Omron CX-Programmer project 新工程 (CX-Programmer 9.73)

# PLC 新PLC1: CPM1(CPM1A) CPU30

## Global symbols (name address type ; comment)
10.00 BOOL  ; KUP
10.01 BOOL  ; KDN
CNT012 BOOL  ; 50

## Program 新程序1 (no task)
; 项目信息： / 这是一个商场中的自动扶梯控制系统，使用欧姆龙 PLC 控制器 CPM1(CPM1A) CPU30 实现。 / 系统通过启动按钮启动扶梯运行，只有在停止按钮未按下时才能启动。 / 操作人员通过上行按钮和下行按钮选择运行方向，上行模式和下行模式不能同时为真。 / 在扶梯运行过程中，操作人员不能手动控制扶梯方向。 / 设备信息： / 系统使用PLC控制器CPM1(CPM1A) CPU30进行控制。 / 硬件包括启动按钮、上行按钮、下行按钮、停止按钮、安全传感器、速度传感器、故障信号输入和报警灯。 / 预期控制： / 系统通过启动按钮和运行使能启动扶梯运行，运行使能由停止按钮2控制。 / 操作人员通过上行按钮和下行按钮选择运行方向，分别激活上行控制或下行控制。 / 上行控制和下行控制通过互锁逻辑设计，尝试避免同时激活。 / 扶梯运行时，安全传感器1-5和速度传感器实时监控状态。 / 安全传感器5检测到异常时，通过计数器记录，若计数器值小于50，设置标志。 / 速度传感器检测到速度异常时，置位速度异常标志。 / 故障信号1-6触发时，置位故障标志1-6。 / 故障信号1触发时，置位故障标志1，记录故障状态。 / 在扶梯运行过程中，方向选择受定时器和标志控制。 / 停止按钮1和停止按钮2可影响扶梯运行，具体逻辑由定时器和内部标志控制。 / 手动/自动切换开关允许操作人员灵活选择控制模式，运行状态输出则向外部设备反馈扶梯运行状态。

### Section 段1

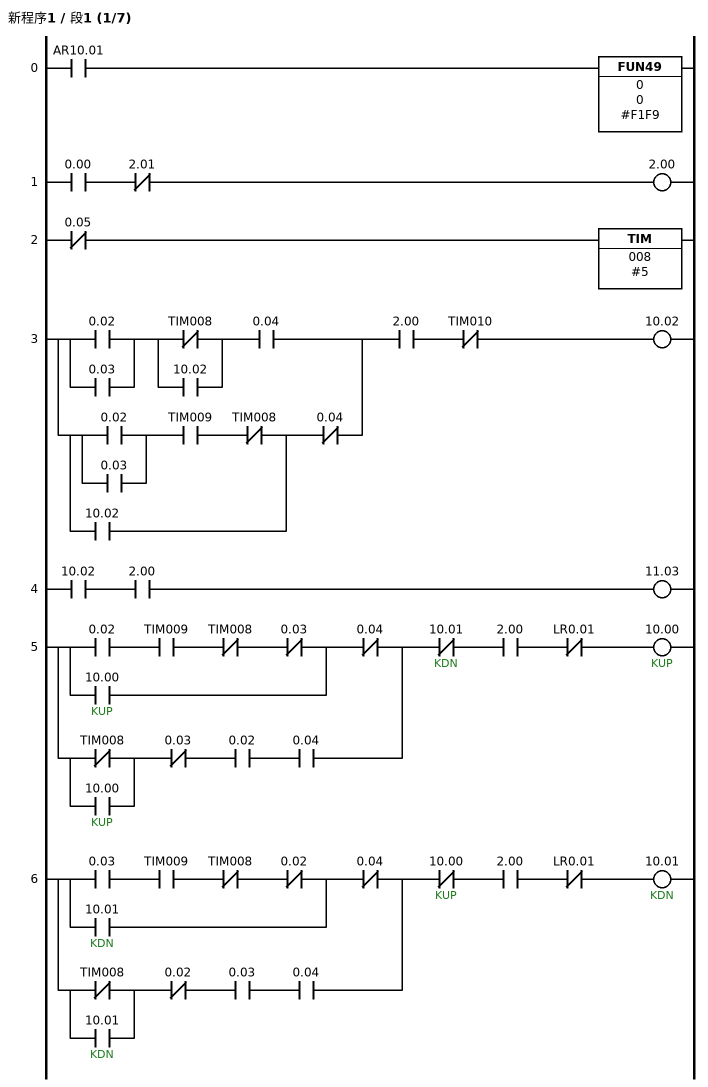
; rung 0
LD AR10.01
FUN49 0 0 #F1F9
; rung 1
LD 0.00
ANDNOT 2.01
OUT 2.00
; rung 2
LDNOT 0.05
TIM 008 #5
; rung 3
LD 0.02
OR 0.03
LDNOT TIM008
OR 10.02
ANDLD
AND 0.04
LD 0.02
OR 0.03
AND TIM009
ANDNOT TIM008
OR 10.02
ANDNOT 0.04
ORLD
AND 2.00
ANDNOT TIM010
OUT 10.02
; rung 4
LD 10.02
AND 2.00
OUT 11.03
; rung 5
LD 0.02
AND TIM009
ANDNOT TIM008
ANDNOT 0.03
OR 10.00  ; KUP
ANDNOT 0.04
LDNOT TIM008
OR 10.00  ; KUP
ANDNOT 0.03
AND 0.02
AND 0.04
ORLD
ANDNOT 10.01  ; KDN
AND 2.00
ANDNOT LR0.01
OUT 10.00  ; KUP
; rung 6
LD 0.03
AND TIM009
ANDNOT TIM008
ANDNOT 0.02
OR 10.01  ; KDN
ANDNOT 0.04
LDNOT TIM008
OR 10.01  ; KDN
ANDNOT 0.02
AND 0.03
AND 0.04
ORLD
ANDNOT 10.00  ; KUP
AND 2.00
ANDNOT LR0.01
OUT 10.01  ; KDN

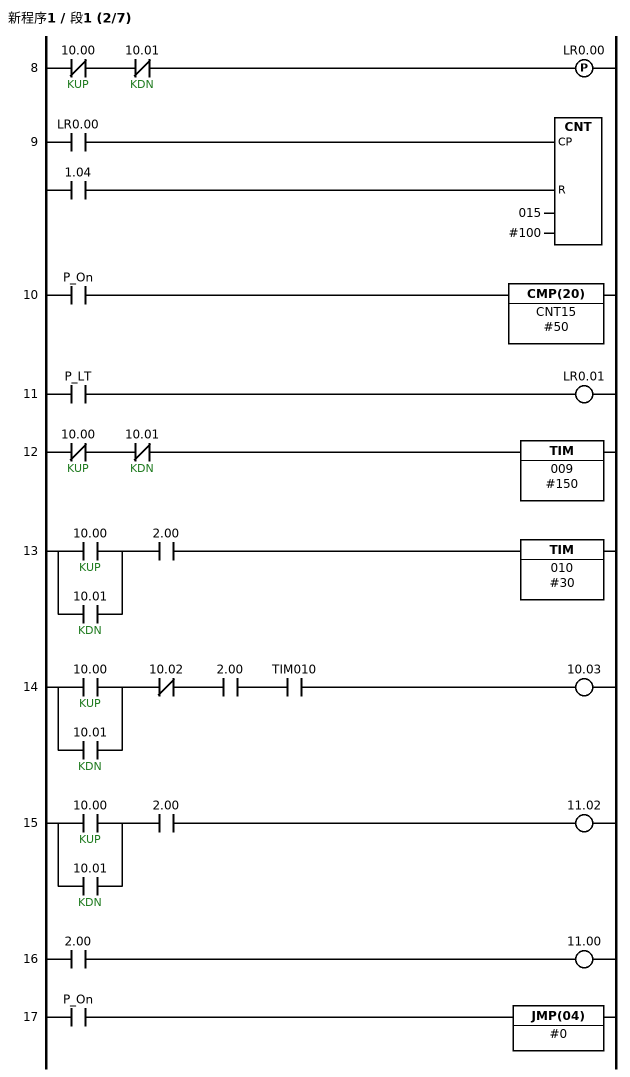
; rung 8
LDNOT 10.00  ; KUP
ANDNOT 10.01  ; KDN
DIFU(13) LR0.00
; rung 9
LD LR0.00
LD 1.04
CNT 015 #100
; rung 10
LD P_On
CMP(20) CNT15 #50
; rung 11
LD P_LT
OUT LR0.01
; rung 12
LDNOT 10.00  ; KUP
ANDNOT 10.01  ; KDN
TIM 009 #150
; rung 13
LD 10.00  ; KUP
OR 10.01  ; KDN
AND 2.00
TIM 010 #30
; rung 14
LD 10.00  ; KUP
OR 10.01  ; KDN
ANDNOT 10.02
AND 2.00
AND TIM010
OUT 10.03
; rung 15
LD 10.00  ; KUP
OR 10.01  ; KDN
AND 2.00
OUT 11.02
; rung 16
LD 2.00
OUT 11.00
; rung 17
LD P_On
JMP(04) #0

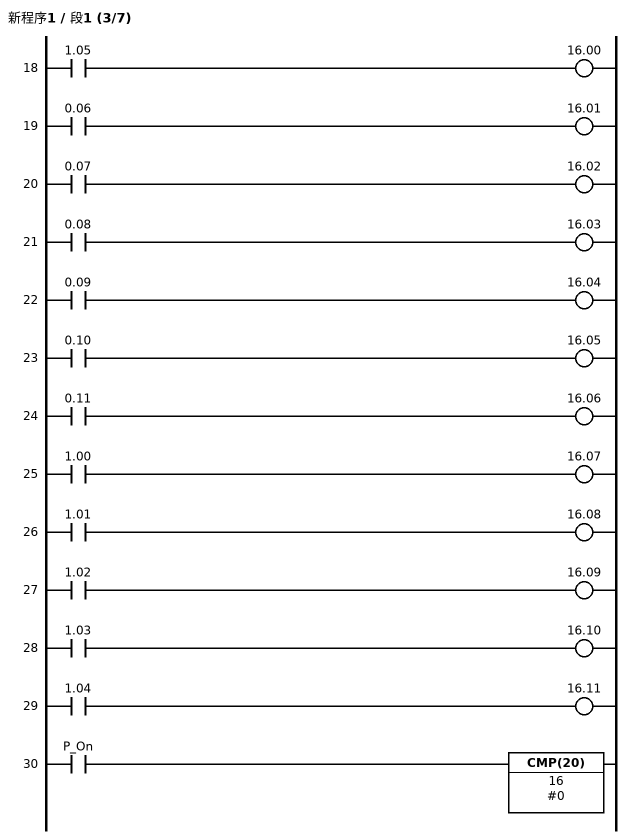
; rung 18
LD 1.05
OUT 16.00
; rung 19
LD 0.06
OUT 16.01
; rung 20
LD 0.07
OUT 16.02
; rung 21
LD 0.08
OUT 16.03
; rung 22
LD 0.09
OUT 16.04
; rung 23
LD 0.10
OUT 16.05
; rung 24
LD 0.11
OUT 16.06
; rung 25
LD 1.00
OUT 16.07
; rung 26
LD 1.01
OUT 16.08
; rung 27
LD 1.02
OUT 16.09
; rung 28
LD 1.03
OUT 16.10
; rung 29
LD 1.04
OUT 16.11
; rung 30
LD P_On
CMP(20) 16 #0

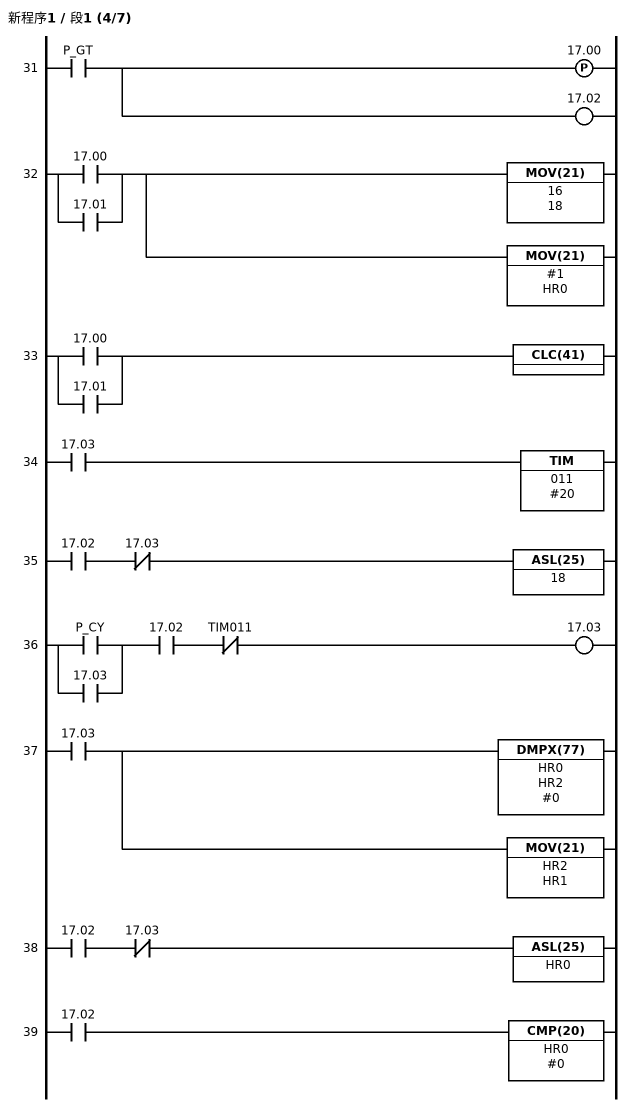
; rung 31
LD P_GT
DIFU(13) 17.00
OUT 17.02
; rung 32
LD 17.00
OR 17.01
MOV(21) 16 18
MOV(21) #1 HR0
; rung 33
LD 17.00
OR 17.01
CLC(41)
; rung 34
LD 17.03
TIM 011 #20
; rung 35
LD 17.02
ANDNOT 17.03
ASL(25) 18
; rung 36
LD P_CY
OR 17.03
AND 17.02
ANDNOT TIM011
OUT 17.03
; rung 37
LD 17.03
DMPX(77) HR0 HR2 #0
MOV(21) HR2 HR1
; rung 38
LD 17.02
ANDNOT 17.03
ASL(25) HR0
; rung 39
LD 17.02
CMP(20) HR0 #0

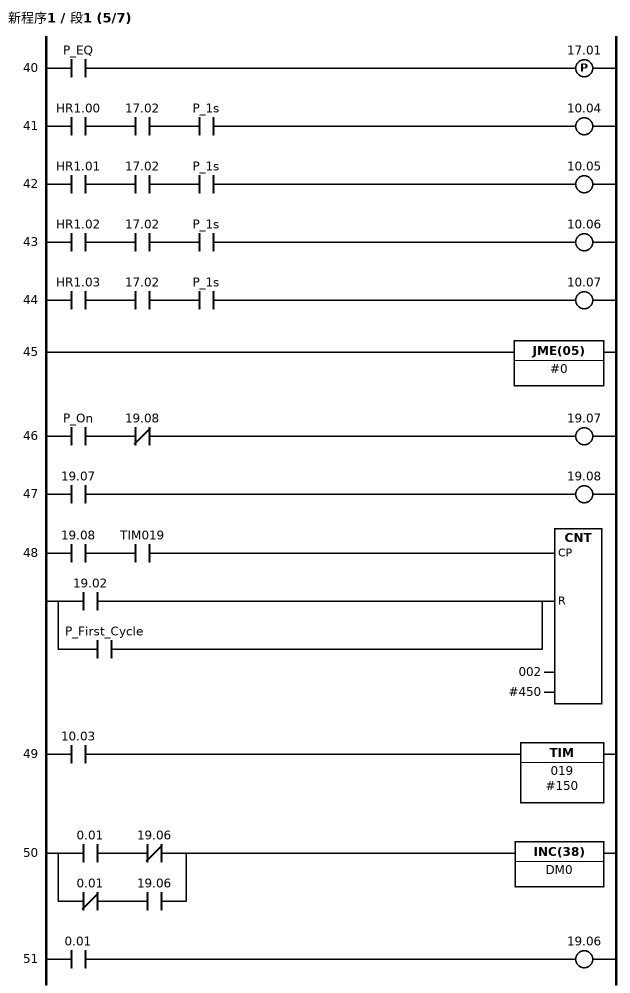
; rung 40
LD P_EQ
DIFU(13) 17.01
; rung 41
LD HR1.00
AND 17.02
AND P_1s
OUT 10.04
; rung 42
LD HR1.01
AND 17.02
AND P_1s
OUT 10.05
; rung 43
LD HR1.02
AND 17.02
AND P_1s
OUT 10.06
; rung 44
LD HR1.03
AND 17.02
AND P_1s
OUT 10.07
; rung 45
JME(05) #0
; rung 46
LD P_On
ANDNOT 19.08
OUT 19.07
; rung 47
LD 19.07
OUT 19.08
; rung 48
LD 19.08
AND TIM019
LD 19.02
OR P_First_Cycle
CNT 002 #450
; rung 49
LD 10.03
TIM 019 #150
; rung 50
LD 0.01
ANDNOT 19.06
LDNOT 0.01
AND 19.06
ORLD
INC(38) DM0
; rung 51
LD 0.01
OUT 19.06

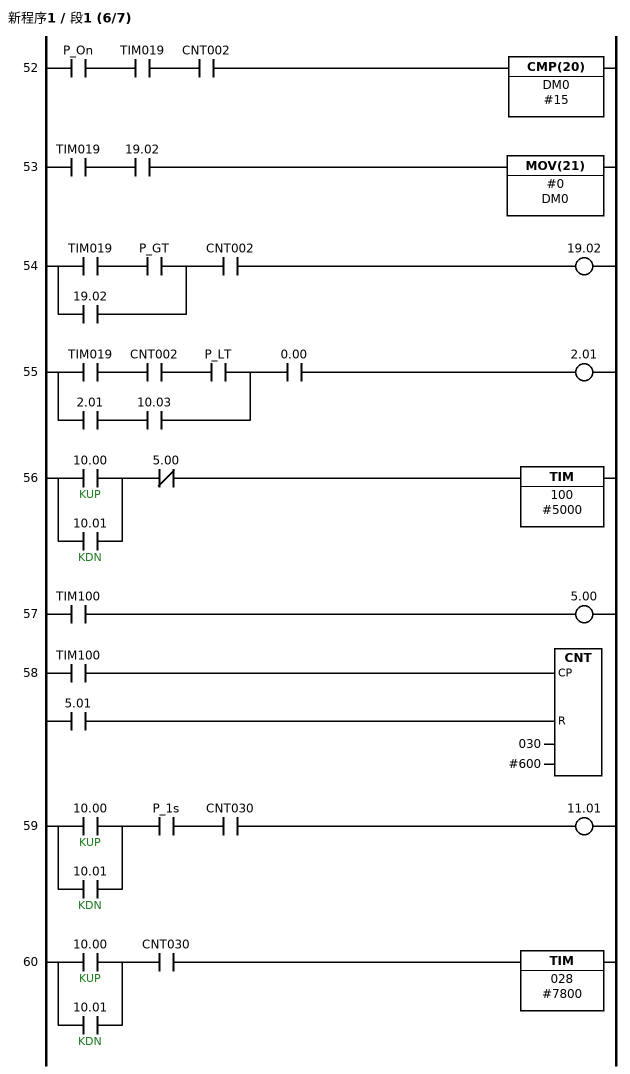
; rung 52
LD P_On
AND TIM019
AND CNT002
CMP(20) DM0 #15
; rung 53
LD TIM019
AND 19.02
MOV(21) #0 DM0
; rung 54
LD TIM019
AND P_GT
OR 19.02
AND CNT002
OUT 19.02
; rung 55
LD TIM019
AND CNT002
AND P_LT
LD 2.01
AND 10.03
ORLD
AND 0.00
OUT 2.01
; rung 56
LD 10.00  ; KUP
OR 10.01  ; KDN
ANDNOT 5.00
TIM 100 #5000
; rung 57
LD TIM100
OUT 5.00
; rung 58
LD TIM100
LD 5.01
CNT 030 #600
; rung 59
LD 10.00  ; KUP
OR 10.01  ; KDN
AND P_1s
AND CNT030
OUT 11.01
; rung 60
LD 10.00  ; KUP
OR 10.01  ; KDN
AND CNT030
TIM 028 #7800

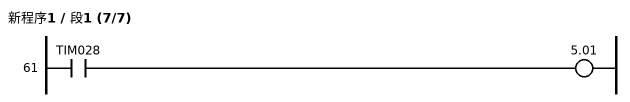
; rung 61
LD TIM028
OUT 5.01
; rung 62
END(01)